// TwinCAT 3 PLC project PLC1
// ProgramVersion: 3.1.4023.0
// libraries:
//   Tc2_Standard, * (Beckhoff Automation GmbH)
//   Tc2_System, * (Beckhoff Automation GmbH)
//   Tc3_Module, * (Beckhoff Automation GmbH)
// project tree:
//   GVLs/ GVL_IHM.TcGVL
//   / PlcTask.TcTTO
//   POUs/ Class Diagram.TcCD (not stored), FB_Robot.TcPOU, FB_System.TcPOU, FB_Wheel.TcPOU, MAIN.TcPOU
// real-time tasks:
//   TASK PlcTask: cycle T#10ms, priority 20, ADS port 350

CONFIGURATION PLC1
    RESOURCE PLC ON TwinCAT3
        TASK PlcTask(INTERVAL := T#10ms, PRIORITY := 20);
        PROGRAM MAIN WITH PlcTask : MAIN;
        PROGRAM MAIN WITH PlcTask : MAIN;
    END_RESOURCE
END_CONFIGURATION

// ---- GVLs/GVL_IHM.TcGVL
{attribute 'qualified_only'}
VAR_GLOBAL
	// Simulation IHM
	StartSystem: BOOL;
	StopSystem: BOOL;

END_VAR

// ---- POUs/MAIN.TcPOU
PROGRAM MAIN
VAR
	fb_System_1: FB_System;
END_VAR

fb_System_1(bStart := GVL_IHM.StartSystem, bStop := GVL_IHM.StopSystem); // FB_System

END_PROGRAM

// ---- POUs/FB_System.TcPOU
FUNCTION_BLOCK FB_System
VAR_INPUT
	bStart: BOOL;
	bStop: BOOL;
END_VAR
VAR_OUTPUT
	bInOperation: BOOL;
END_VAR
VAR
	fb_Robot_1: FB_Robot;
	fb_Robot_2: FB_Robot;
	SR_1: SR;
END_VAR

fb_Robot_2(bEnable := SR_1.Q1); // FB_Robot
bInOperation := SR_1.Q1;
SR_1(SET1 := bStart, RESET := bStop); // SR
fb_Robot_1(bEnable := SR_1.Q1); // FB_Robot

END_FUNCTION_BLOCK

// ---- POUs/FB_Robot.TcPOU
FUNCTION_BLOCK FB_Robot
VAR_INPUT
	bEnable: BOOL;
	bReset: BOOL;
END_VAR
VAR_OUTPUT
	bBusy: BOOL;
	bError: BOOL;
END_VAR
VAR
	fb_Wheel_1: FB_Wheel;
	fb_Wheel_2: FB_Wheel;
	fb_Wheel_3: FB_Wheel;
	fb_Wheel_4: FB_Wheel;
END_VAR

fb_Wheel_1(); // FB_Wheel
// bEnable: input not connected

END_FUNCTION_BLOCK

// ---- POUs/FB_Wheel.TcPOU
FUNCTION_BLOCK FB_Wheel
VAR_INPUT
END_VAR
VAR_OUTPUT
END_VAR
VAR
END_VAR

PROPERTY Speed : real
GET
END_GET
SET
END_SET
END_PROPERTY

END_FUNCTION_BLOCK
